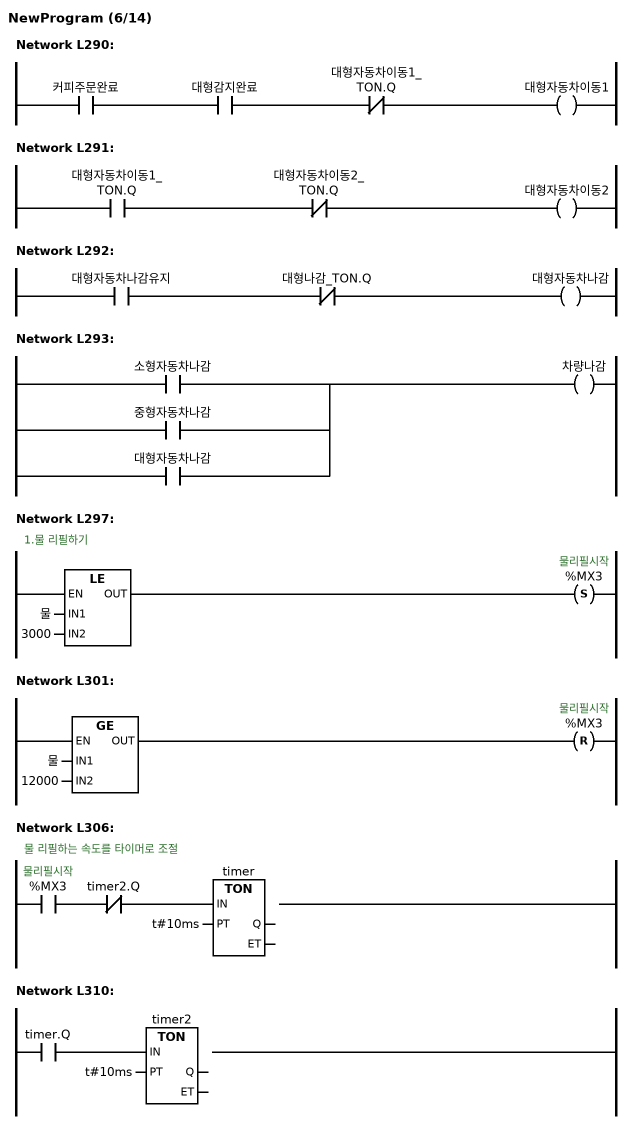
(* [picture p24: NewProgram rungs L290-L310] *)
(* Rung L290 *)
대형자동차이동1 := 커피주문완료 AND 대형감지완료 AND NOT 대형자동차이동1_TON.Q;
(* Rung L291 *)
대형자동차이동2 := 대형자동차이동1_TON.Q AND NOT 대형자동차이동2_TON.Q;
(* Rung L292 *)
대형자동차나감 := 대형자동차나감유지 AND NOT 대형나감_TON.Q;
(* Rung L293 *)
차량나감 := 소형자동차나감 OR 중형자동차나감 OR 대형자동차나감;
(* 1.물 리필하기 *)
(* Rung L297 *)
IF 물 <= 3000 THEN %MX3 := TRUE; END_IF;
(* Rung L301 *)
IF 물 >= 12000 THEN %MX3 := FALSE; END_IF;
(* 물 리필하는 속도를 타이머로 조절 *)
(* Rung L306 *)
timer(IN := %MX3 AND NOT timer2.Q, PT := t#10ms);
(* Rung L310 *)
timer2(IN := timer.Q, PT := t#10ms);

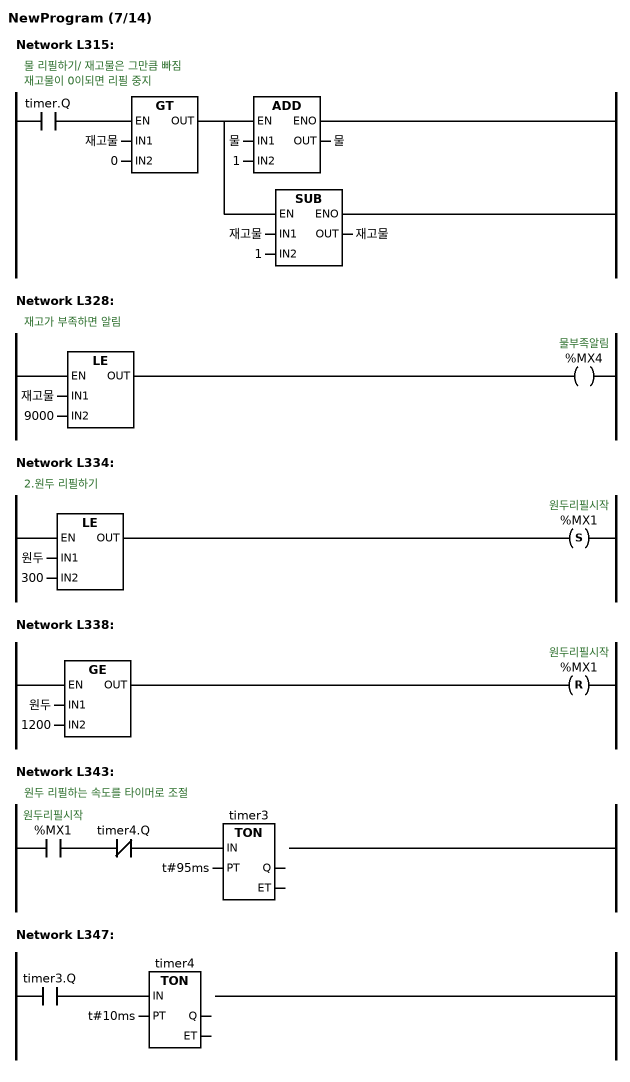
(* 물 리필하기/ 재고물은 그만큼 빠짐 *)
(* 재고물이 0이되면 리필 중지 *)
(* Rung L315 *)
IF timer.Q THEN _t6 := 재고물 > 0; END_IF;
IF _t6 THEN
    물 := 물 + 1;
    재고물 := 재고물 - 1;
END_IF;
(* 재고가 부족하면 알림 *)
(* Rung L328 *)
%MX4 := 재고물 <= 9000;
(* 2.원두 리필하기 *)
(* Rung L334 *)
IF 원두 <= 300 THEN %MX1 := TRUE; END_IF;
(* Rung L338 *)
IF 원두 >= 1200 THEN %MX1 := FALSE; END_IF;
(* 원두 리필하는 속도를 타이머로 조절 *)
(* Rung L343 *)
timer3(IN := %MX1 AND NOT timer4.Q, PT := t#95ms);
(* Rung L347 *)
timer4(IN := timer3.Q, PT := t#10ms);

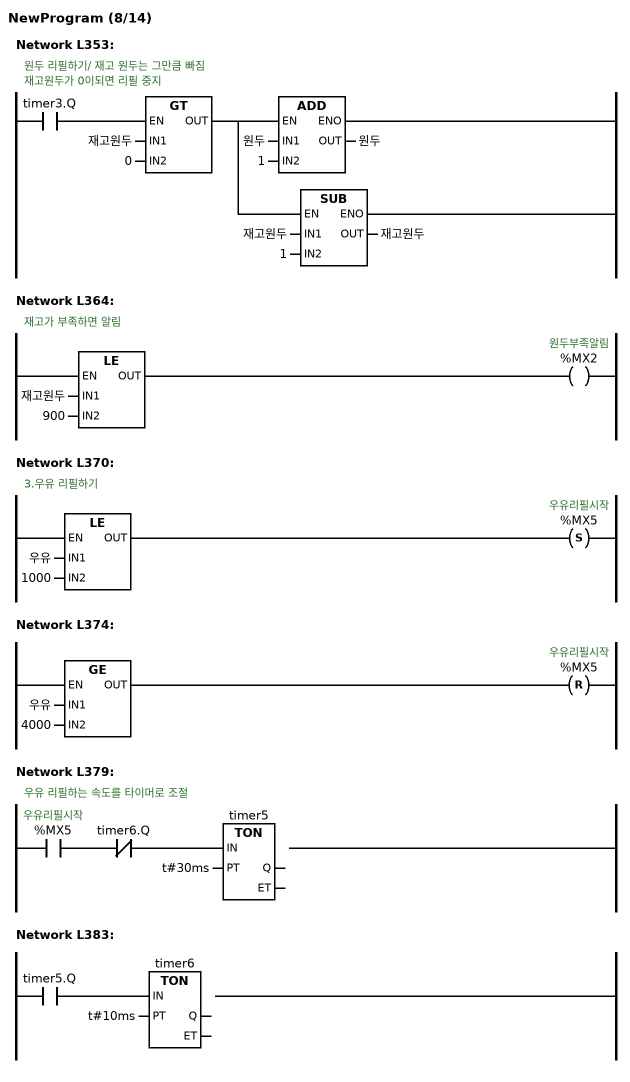
(* 원두 리필하기/ 재고 원두는 그만큼 빠짐 *)
(* 재고원두가 0이되면 리필 중지 *)
(* Rung L353 *)
IF timer3.Q THEN _t7 := 재고원두 > 0; END_IF;
IF _t7 THEN
    원두 := 원두 + 1;
    재고원두 := 재고원두 - 1;
END_IF;
(* 재고가 부족하면 알림 *)
(* Rung L364 *)
%MX2 := 재고원두 <= 900;
(* 3.우유 리필하기 *)
(* Rung L370 *)
IF 우유 <= 1000 THEN %MX5 := TRUE; END_IF;
(* Rung L374 *)
IF 우유 >= 4000 THEN %MX5 := FALSE; END_IF;
(* 우유 리필하는 속도를 타이머로 조절 *)
(* Rung L379 *)
timer5(IN := %MX5 AND NOT timer6.Q, PT := t#30ms);
(* Rung L383 *)
timer6(IN := timer5.Q, PT := t#10ms);

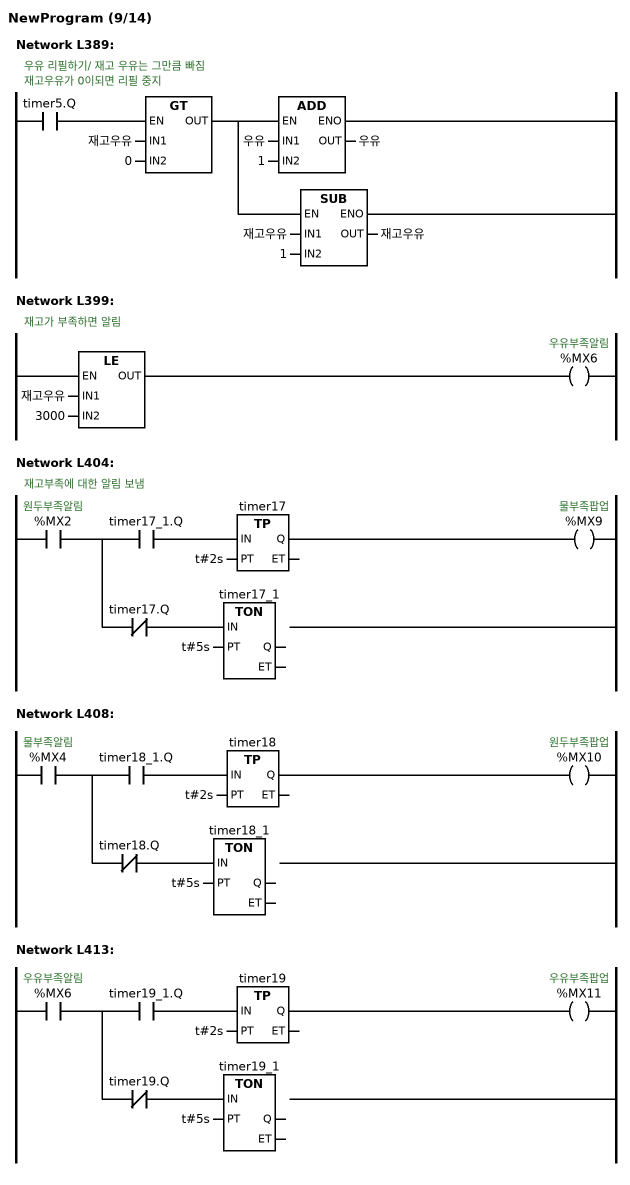
(* 우유 리필하기/ 재고 우유는 그만큼 빠짐 *)
(* 재고우유가 0이되면 리필 중지 *)
(* Rung L389 *)
IF timer5.Q THEN _t8 := 재고우유 > 0; END_IF;
IF _t8 THEN
    우유 := 우유 + 1;
    재고우유 := 재고우유 - 1;
END_IF;
(* 재고가 부족하면 알림 *)
(* Rung L399 *)
%MX6 := 재고우유 <= 3000;
(* 재고부족에 대한 알림 보냄 *)
(* Rung L404 *)
timer17(IN := %MX2 AND timer17_1.Q, PT := t#2s);
%MX9 := timer17.Q;
timer17_1(IN := %MX2 AND NOT timer17.Q, PT := t#5s);
(* Rung L408 *)
timer18(IN := %MX4 AND timer18_1.Q, PT := t#2s);
%MX10 := timer18.Q;
timer18_1(IN := %MX4 AND NOT timer18.Q, PT := t#5s);
(* Rung L413 *)
timer19(IN := %MX6 AND timer19_1.Q, PT := t#2s);
%MX11 := timer19.Q;
timer19_1(IN := %MX6 AND NOT timer19.Q, PT := t#5s);

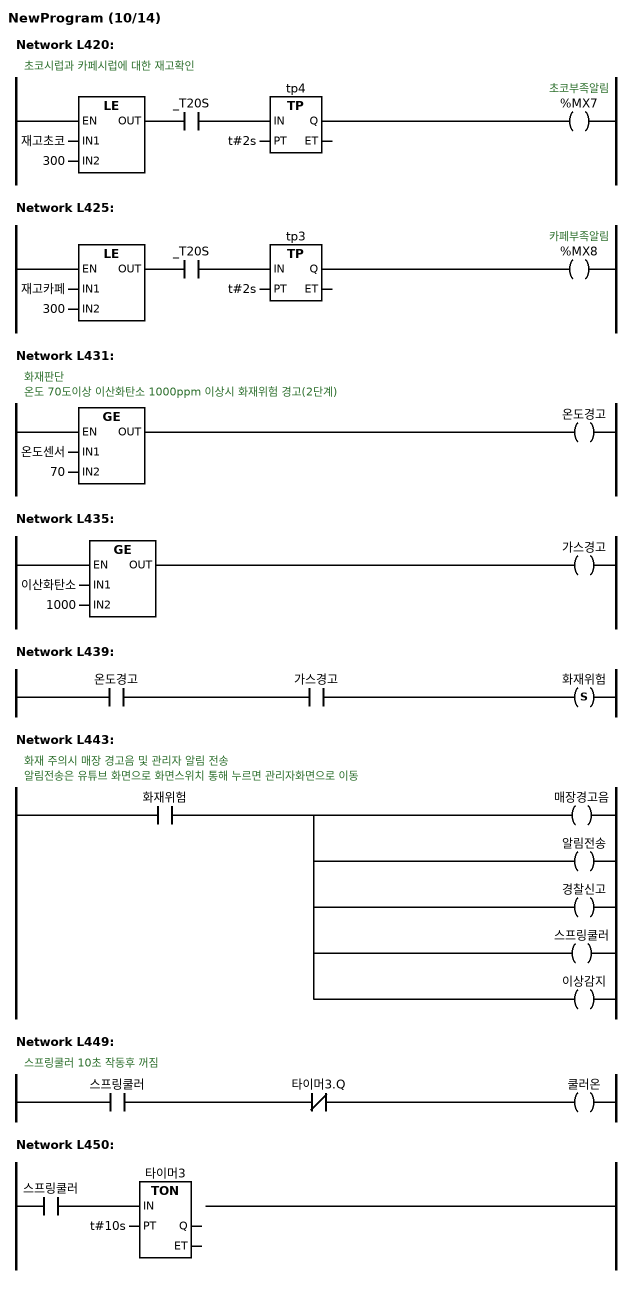
(* 초코시럽과 카페시럽에 대한 재고확인 *)
(* Rung L420 *)
tp4(IN := (재고초코 <= 300) AND _T20S, PT := t#2s);
%MX7 := tp4.Q;
(* Rung L425 *)
tp3(IN := (재고카페 <= 300) AND _T20S, PT := t#2s);
%MX8 := tp3.Q;
(* 화재판단 *)
(* 온도 70도이상 이산화탄소 1000ppm 이상시 화재위험 경고(2단계) *)
(* Rung L431 *)
온도경고 := 온도센서 >= 70;
(* Rung L435 *)
가스경고 := 이산화탄소 >= 1000;
(* Rung L439 *)
IF 온도경고 AND 가스경고 THEN 화재위험 := TRUE; END_IF;
(* 화재 주의시 매장 경고음 및 관리자 알림 전송 *)
(* 알림전송은 유튜브 화면으로 화면스위치 통해 누르면 관리자화면으로 이동 *)
(* Rung L443 *)
매장경고음 := 화재위험;
알림전송 := 화재위험;
경찰신고 := 화재위험;
스프링쿨러 := 화재위험;
이상감지 := 화재위험;
(* 스프링쿨러 10초 작동후 꺼짐 *)
(* Rung L449 *)
쿨러온 := 스프링쿨러 AND NOT 타이머3.Q;
(* Rung L450 *)
타이머3(IN := 스프링쿨러, PT := t#10s);

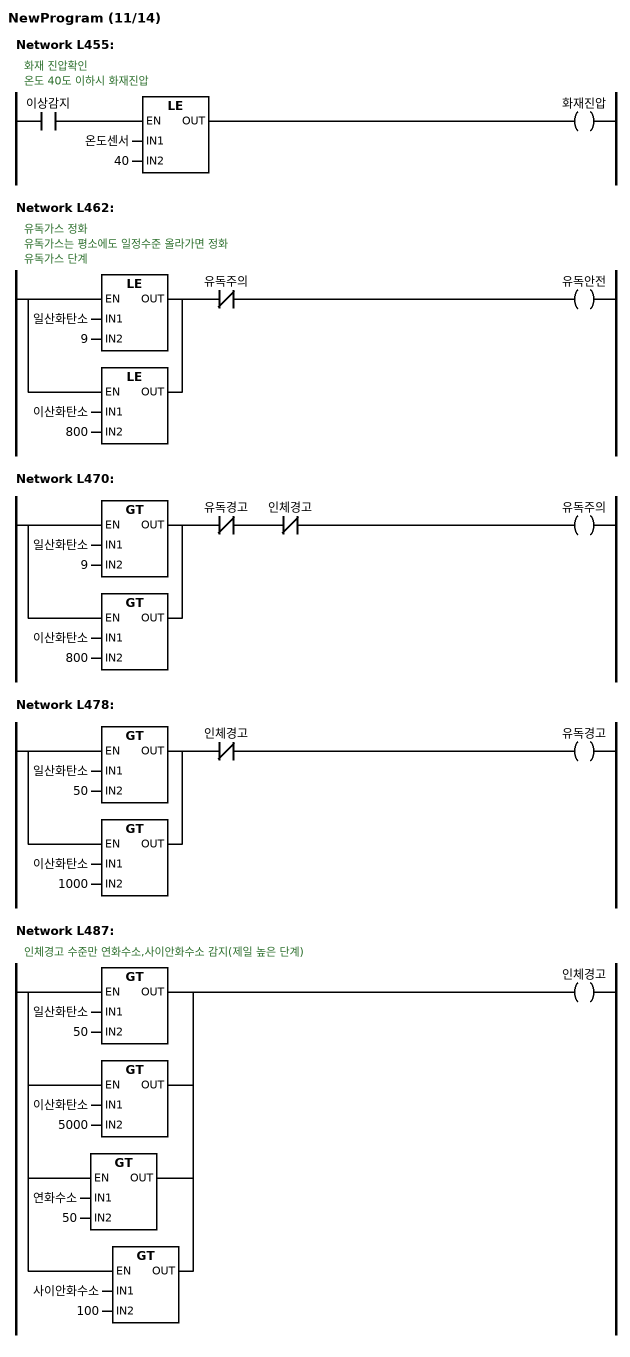
(* 화재 진압확인 *)
(* 온도 40도 이하시 화재진압 *)
(* Rung L455 *)
IF 이상감지 THEN _t9 := 온도센서 <= 40; END_IF;
화재진압 := _t9;
(* 유독가스 정화 *)
(* 유독가스는 평소에도 일정수준 올라가면 정화 *)
(* 유독가스 단계 *)
(* Rung L462 *)
유독안전 := ((일산화탄소 <= 9) OR (이산화탄소 <= 800)) AND NOT 유독주의;
(* Rung L470 *)
유독주의 := ((일산화탄소 > 9) OR (이산화탄소 > 800)) AND NOT 유독경고 AND NOT 인체경고;
(* Rung L478 *)
유독경고 := ((일산화탄소 > 50) OR (이산화탄소 > 1000)) AND NOT 인체경고;
(* 인체경고 수준만 연화수소,사이안화수소 감지(제일 높은 단계) *)
(* Rung L487 *)
인체경고 := (일산화탄소 > 50) OR (이산화탄소 > 5000) OR (연화수소 > 50) OR (사이안화수소 > 100);

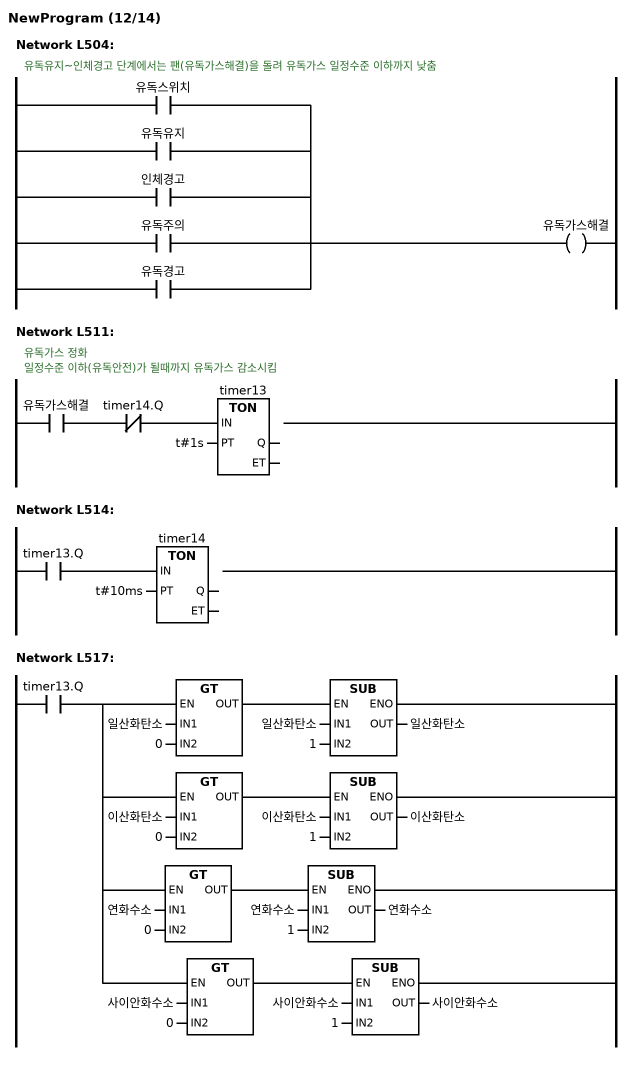
(* 유독유지~인체경고 단계에서는 팬(유독가스해결)을 돌려 유독가스 일정수준 이하까지 낮춤 *)
(* Rung L504 *)
유독가스해결 := 유독스위치 OR 유독유지 OR 인체경고 OR 유독주의 OR 유독경고;
(* 유독가스 정화 *)
(* 일정수준 이하(유독안전)가 될때까지 유독가스 감소시킴 *)
(* Rung L511 *)
timer13(IN := 유독가스해결 AND NOT timer14.Q, PT := t#1s);
(* Rung L514 *)
timer14(IN := timer13.Q, PT := t#10ms);
(* Rung L517 *)
IF timer13.Q THEN _t10 := 일산화탄소 > 0; END_IF;
IF _t10 THEN 일산화탄소 := 일산화탄소 - 1; END_IF;
IF timer13.Q THEN _t11 := 이산화탄소 > 0; END_IF;
IF _t11 THEN 이산화탄소 := 이산화탄소 - 1; END_IF;
IF timer13.Q THEN _t12 := 연화수소 > 0; END_IF;
IF _t12 THEN 연화수소 := 연화수소 - 1; END_IF;
IF timer13.Q THEN _t13 := 사이안화수소 > 0; END_IF;
IF _t13 THEN 사이안화수소 := 사이안화수소 - 1; END_IF;

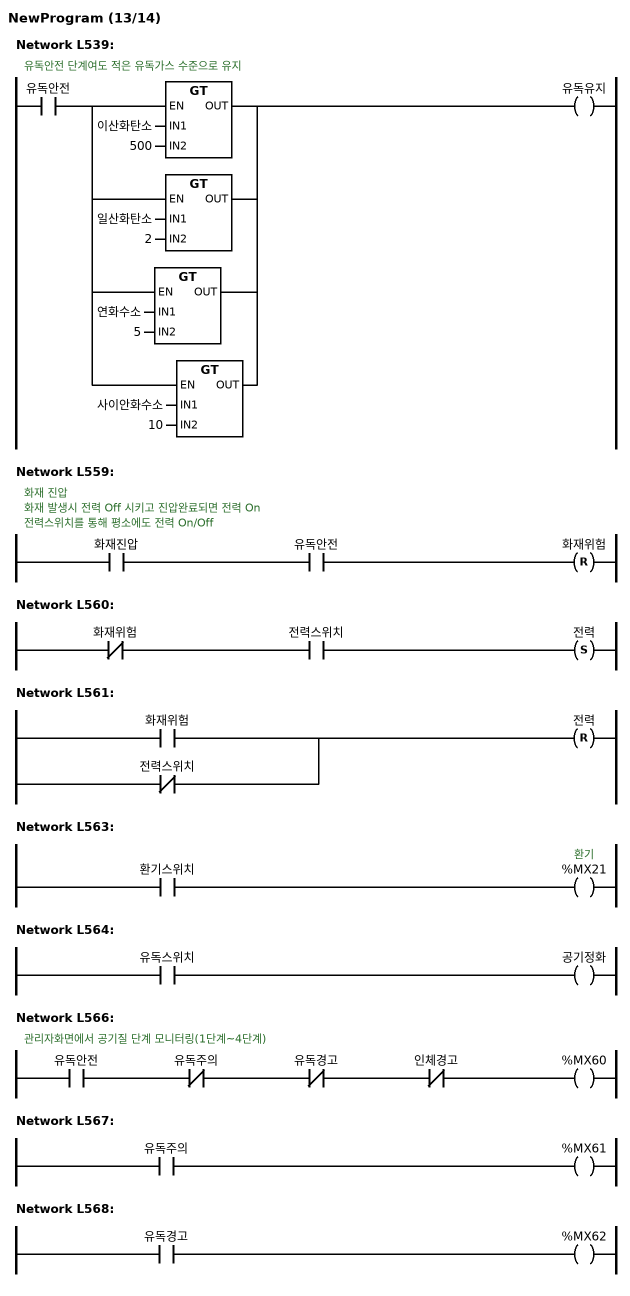
(* 유독안전 단계여도 적은 유독가스 수준으로 유지 *)
(* Rung L539 *)
IF 유독안전 THEN
    _t14 := 이산화탄소 > 500;
    _t15 := 일산화탄소 > 2;
    _t16 := 연화수소 > 5;
    _t17 := 사이안화수소 > 10;
END_IF;
유독유지 := _t14 OR _t15 OR _t16 OR _t17;
(* 화재 진압 *)
(* 화재 발생시 전력 Off 시키고 진압완료되면 전력 On *)
(* 전력스위치를 통해 평소에도 전력 On/Off *)
(* Rung L559 *)
IF 화재진압 AND 유독안전 THEN 화재위험 := FALSE; END_IF;
(* Rung L560 *)
IF NOT 화재위험 AND 전력스위치 THEN 전력 := TRUE; END_IF;
(* Rung L561 *)
IF 화재위험 OR NOT 전력스위치 THEN 전력 := FALSE; END_IF;
(* Rung L563 *)
%MX21 := 환기스위치;
(* Rung L564 *)
공기정화 := 유독스위치;
(* 관리자화면에서 공기질 단계 모니터링(1단계~4단계) *)
(* Rung L566 *)
%MX60 := 유독안전 AND NOT 유독주의 AND NOT 유독경고 AND NOT 인체경고;
(* Rung L567 *)
%MX61 := 유독주의;
(* Rung L568 *)
%MX62 := 유독경고;

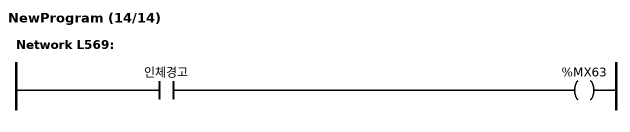
(* Rung L569 *)
%MX63 := 인체경고;
END_PROGRAM